TYPE ST_SEARCH_SHAPE :
STRUCT
	aCenterPoint			: TcVnPoint2_REAL;
	nHeight					: REAL;
	nWidth					: REAL;
END_STRUCT
END_TYPE

(* stored: Version 1.1.0.1, ProductVersion 3.1.4024.12
   DUT ST_SEARCH_SHAPE: Id {52936523-c7e3-4565-a0c6-b4732f1ba4f2} *)
